(* PLC project Sin nombre, Desconocido Sin nombre 1 *)
(* stored: creationDateTime 2025-09-25T16:50:19, modificationDateTime 2025-09-25T17:07:33 *)

PROGRAM RA23
  VAR_INPUT
    B1 : BOOL;
    B2 : BOOL;
    B3 : BOOL;
  END_VAR
  VAR_OUTPUT
    H1 : BOOL;
    H2 : BOOL;
    H6 : BOOL;
    H3 : BOOL;
    H4 : BOOL;
    H5 : BOOL;
    Pump : BOOL;
    V1 : BOOL;
    V2 : BOOL;
  END_VAR

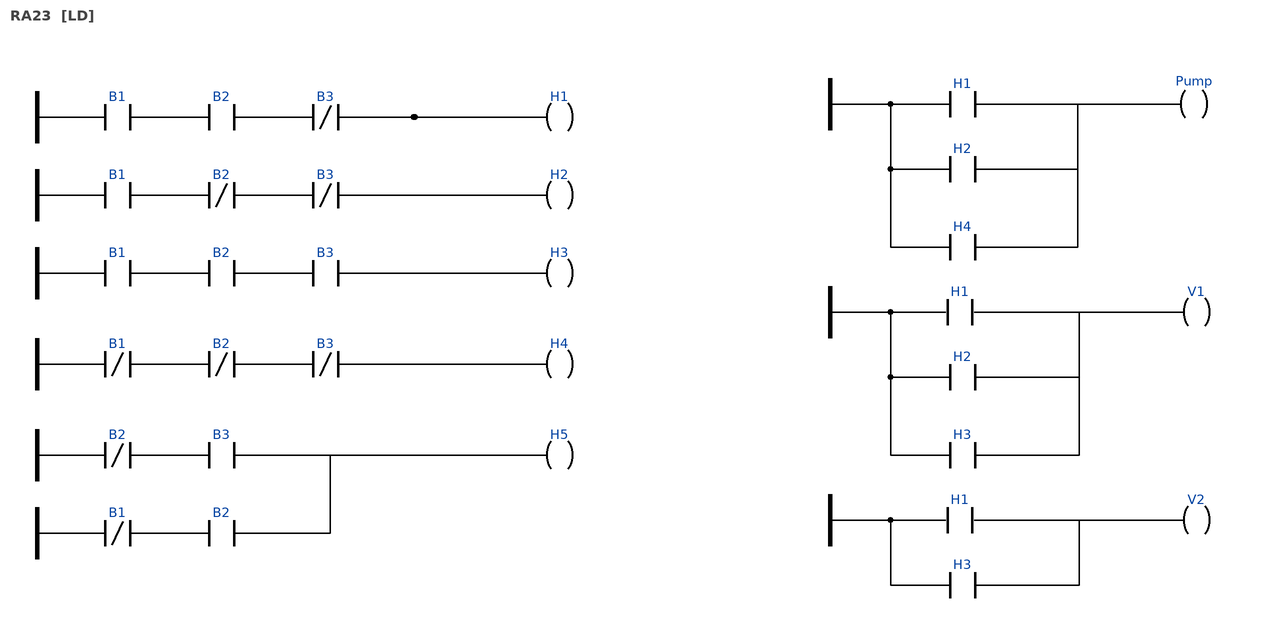
(* LD diagram, written out as Structured Text *)
H5 := NOT B2 AND B3 OR NOT B1 AND B2;
H4 := NOT B1 AND NOT B2 AND NOT B3;
H3 := B1 AND B2 AND B3;
H2 := B1 AND NOT B2 AND NOT B3;
H1 := B1 AND B2 AND NOT B3;
Pump := H1 OR H2 OR H4;
V1 := H1 OR H3 OR H2;
V2 := H1 OR H3;
END_PROGRAM

CONFIGURATION Config0
  RESOURCE Res0 ON PLC
    TASK task0(INTERVAL := T#20ms, PRIORITY := 0);
    PROGRAM instance0 WITH task0 : RA23;
  END_RESOURCE
END_CONFIGURATION
